Fanuc KAREL source: DAQ_UNREG.kl

PROGRAM T
%NOLOCKGROUP
VAR
 v0 : INTEGER
 v1 : INTEGER
BEGIN
 DAQ_UNREG(v0, v1)
END T
